FUNCTION_BLOCK FB_QuantityINTPublic EXTENDS FB_FalliblePublic IMPLEMENTS I_QuantityINTPublic
VAR
    {attribute 'pytmc' := '
        pv: Value
        io: io
        field: DESC Value of quantity.
    '}
    nValue : INT;

    {attribute 'pytmc' := '
        pv: Units
        io: io
        field: DESC Units of quantity.
    '}
    sUnits : T_MaxString;
END_VAR


METHOD Copy
VAR_INPUT
    QuantityToCopy : I_QuantityINT;
END_VAR

Val := QuantityToCopy.Val;
Units := QuantityToCopy.Units;

IF QuantityToCopy.GetError() THEN
    SetError(Msg := QuantityToCopy.GetErrorMsg());
ELSE
    ClearError();
END_IF
END_METHOD


METHOD FB_Init: BOOL
VAR_INPUT
    bInitRetains: BOOL; // TRUE: the retain variables are initialized (reset warm / reset cold)
    bInCopyCode: BOOL;  // TRUE: the instance will be copied to the copy code afterward (online change)

    Units : T_MaxString;
END_VAR

THIS^.Units := Units;
END_METHOD


PROPERTY Units : T_MaxString
GET

Units := sUnits;
END_GET
SET

sUnits := Units;
END_SET
END_PROPERTY


PROPERTY Val : INT
GET

Val := nValue;
END_GET
SET

nValue := Val;
END_SET
END_PROPERTY

END_FUNCTION_BLOCK

(* stored: Version 1.1.0.1
   POU FB_QuantityINTPublic: Id {8e2c99df-d649-4bfc-a956-baf4a7b6ac0e}, SpecialFunc None
   Method Copy: Id {6f88bde4-c6bd-4a44-8b41-302e399f8a90}
   Method FB_Init: Id {5707d2e2-0fa5-4325-b044-341311ed4385}
   Property Units: Id {2a0cdbe1-dec3-4f78-bd70-dbba6b5e1c62}
   Get Get: Id {1b9b5d2f-ef6a-4d6b-8fc0-e64e5a287de1}
   Set Set: Id {4d927f6e-373f-455c-b26c-454373e8531c}
   Property Val: Id {da39bdea-8128-4ea2-a0e8-acce7d4fd43e}
   Get Get: Id {204b559b-b427-4ca6-903c-ea60f8c99380}
   Set Set: Id {a54ae9af-7b84-4183-a8c7-57a17fa9c929} *)
